Staubli VAL3: start.pgx

program start()
begin
  call ex12()
end
